// TIA Portal V20 export
// export: Created 2026-08-13T15:18:03.6792671Z, ExportSetting WithDefaults, DisplayName Totally Integrated Automation Portal, DisplayVersion V20 Update 5, DisplayName TIA Portal Openness, DisplayVersion V20 Update 4, DisplayName TIA Portal Version Control Interface, DisplayVersion V20 Update 5, DisplayName SINAMICS Startdrive Advanced, DisplayVersion V20, DisplayName SINAMICS DCC, DisplayVersion V20, DisplayName SINAMICS Startdrive G130, G150, S120, S150, SINAMICS MV, G220, S200, S210, DisplayVersion V20, DisplayName SINAMICS Startdrive G110M, G120, G120C, G120D, G120P, G115D, DisplayVersion V20, DisplayName STEP 7 Professional, DisplayVersion V20 Update 5, DisplayName STEP 7 Safety, DisplayVersion V20 Update 2, DisplayName WinCC Basic/Comfort/Advanced, DisplayVersion V20 Update 5, DisplayName WinCC Unified, DisplayVersion V20 Update 5
DATA_BLOCK "iDB_PusherControl"   // DB10
VERSION : 0.1
// stored: AutoNumber true, DBAccessibleFromOPCUA true, InstanceOfName FB_PusherControl, InstanceOfType FB
"FB_PusherControl"
   // VAR RETAIN
   //    IO { S7_SetPoint := 'True'} : "UDT_PusherIO";
   // END_VAR
   // VAR
   //    CycleRequest : Bool;
   //    JogDemand : Bool;
   //    ReparkRequest : Bool;
   //    LaunchRequest : Bool;
   //    CycleAbort : Bool;
   //    EndTravelTimeoutMS : DInt;
   //    ParkedTimeoutMS : DInt;
   //    EndTravelHoldTimeMS : DInt;
   //    PumpRunOnTimeMS : DInt;
   //    JogWarningTimeMS : DInt;
   //    PressureTripConfirmTimeMS : DInt;
   //    PressureClearResumeDelayMS : DInt;
   //    PressureConfirmTimer { S7_SetPoint := 'True'} : TON_TIME;
   //    PressureClearTimer { S7_SetPoint := 'True'} : TON_TIME;
   //    PressureHold : Bool;
   //    PressureConfirmEdge : Bool;
   //    PressureConfirmEdgeMem : Bool;
   //    PressureTripCount : Int;
   //    EndTravelTimer { S7_SetPoint := 'True'} : TON_TIME;
   //    HoldTimer { S7_SetPoint := 'True'} : TON_TIME;
   //    ParkedTimer { S7_SetPoint := 'True'} : TON_TIME;
   //    JogPreStartTimer { S7_SetPoint := 'True'} : TON_TIME;
   //    ExtendDemand : Bool;
   //    RetractDemand : Bool;
   //    PumpDemand : Bool;
   //    PumpEverDemanded : Bool;
   //    PumpRunOnTimer { S7_SetPoint := 'True'} : TON_TIME;
   // END_VAR
BEGIN
END_DATA_BLOCK
